FUNCTION_BLOCK FB_HomeableAxis EXTENDS FB_Axis
VAR_INPUT
END_VAR
VAR_OUTPUT
END_VAR
VAR
	fbMcHome		: MC_Home;				// FB to home axis
	bDoHoming		:	BOOL; //do action 1 variable
	piHomeSensor	: FB_Input;
END_VAR

(*
	- Version: V2.0
	- Modified: SOHN
	- Time: 20/10/2021
	- Description: Change bHomeSensor into FB_Input: piHomeSensor so that fbHMI can append input. Modify Stop() 
	- Comment: May the moral be with you!!
*)

	IF bFirstCycle THEN
		piHomeSensor.Description := 'Home Detector';
	END_IF

	bHomingable := TRUE;
	bDoHoming := FALSE;
	Super^();

METHOD Home : BOOL // Start axis homing
VAR_INPUT
END_VAR
IF iStepGeneral = 30 THEN
	iStepGeneral := 40;
END_IF

bDoHoming := TRUE;

//Method output
	Home := (iStepGeneral = 50);
END_METHOD

PROPERTY HomeDetector : I_Input
GET
HomeDetector := piHomeSensor;
END_GET
END_PROPERTY

METHOD Reset : BOOL
VAR_INPUT
END_VAR
fbMcHome(			Execute	:= FALSE,
					Axis 	:= AxisRef);
SUPER^.Reset();
END_METHOD

METHOD PROTECTED StateAborting : BOOL
VAR_INPUT
END_VAR
bInitialized := FALSE;
CASE iStepAborting OF
	0: 
		fbMcHome(			Execute	:= FALSE,
							Axis 	:= AxisRef);
END_CASE
Super^.StateAborting();
END_METHOD

METHOD PROTECTED StateHoming : BOOL // Unit is performing action 1
VAR_INPUT
END_VAR
IF NOT fbMcHome.Error THEN // no error behavior

//Home
	fbMcHome(		Execute 	:= TRUE,
					Axis		:= AxisRef,
					HomingMode	:= MC_DefaultHoming,
					bCalibratioNCam		:= piHomeSensor.Value);
	IF fbMcHome.Done THEN
		iStepGeneral := 50;
		fbMcHome(	Execute 	:= FALSE,
					Axis		:= AxisRef,
					HomingMode	:= MC_DefaultHoming,
					bCalibratioNCam		:= piHomeSensor.Value);
	END_IF

ELSE // error behavior
	fbMcHome(		Execute 	:= FALSE,
					Axis		:= AxisRef,
					HomingMode	:= MC_DefaultHoming,
					bCalibratioNCam		:= piHomeSensor.Value);
					
	bError		:= TRUE;
	iErrorID 	:= fbMcHome.ErrorID;
END_IF
END_METHOD

METHOD PROTECTED StateHomingDone : BOOL // Unit has finished action 1, waiting for release of the request
VAR_INPUT
END_VAR
//do something if necessary
IF NOT bDoHoming THEN
	iStepGeneral := 30;
END_IF
END_METHOD

METHOD PROTECTED StateMachine : BOOL // Sate machien of unit
VAR_INPUT
END_VAR

VAR
	StateAction6Done: INT;
END_VAR
//State machine						   
	CASE iStepGeneral OF
		40: //homing
			Enable(TRUE);
			StateHoming();
			
		50: //Homing done
			Enable(TRUE);
			StateHomingDone();
	END_CASE
	
Super^.StateMachine();
END_METHOD

END_FUNCTION_BLOCK

(* stored: Version 1.1.0.1, ProductVersion 3.1.4024.9
   POU FB_HomeableAxis: Id {e39a638c-b17e-40f3-9c35-4e2ad79e6951}, SpecialFunc None
   Method Home: Id {0a754339-1164-4436-ad14-b08d812d6ef7}
   Property HomeDetector: Id {b1678fde-d5c5-4bee-89e9-61ac5bcbb9f3}
   Get Get: Id {4104d17e-3499-4872-8127-e08b84e4e8e0}
   Method Reset: Id {e24f404d-f8db-4b50-b088-6da77ea60e28}
   Method StateAborting: Id {ccc02e71-3a1b-430a-86af-124c3136c9a8}
   Method StateHoming: Id {ad33bc9f-1bc2-46f2-a3f0-c2c3215e843e}
   Method StateHomingDone: Id {5818cf0e-c1af-457a-ba34-8715e4be5345}
   Method StateMachine: Id {794a65f3-bf1c-47dd-8df6-0e8c470b0964} *)
